(*
Nazwa:			FB_MoveRegister
Opis:			Blok przesuniecia rejestru formatek
Wersja:			v0.3 		
Data:			2018-11-16
Autor:			DP
Urzadzenia:		 
Konfiguracja:	
Info:
- Są dwa rejestry, wejściowy i wyjsciowy (struktury)
- Jezeli rejestr ma np. 6 elementów to za kazdym razem po wykryciu trigera program będzie
	1 wejściowy przesuwał na 1 wolny (nie ma formatki) wyjściowy
	kasował 1 rejestr wejściowy
	przesuwal rejetr wejsciowy 2 na 1(przeniesiony i skasowany), 3 na 2, 4 na 3, 5 na 4, 6 na 5 i kasowal 6wejsciowy
	tym sposobem po 6 trigerach caly rejestr wejsciowy powinien być na wyjsciowym
	np po 3 trigerach na wyjsciowym powinny byc zajete 1 do 3 i na wejsciowym 1 do 3
Błędy:
1 - nie wyszło z pętli for
2 - formatka już jest w rejestrze
Uwagi:
- 
Zmiany:
2018-09-18 Dodano sprawdzanie nasadek
2018-06-14 DP Pierwsza wersja
*)

FUNCTION_BLOCK FB_MoveRegister
VAR_INPUT
	bFirstCycle:BOOL;					//Pierwszy cykl, zeby na początku nie wykrywało zbocza opadającego
	bTrigger :BOOL;						// Przesuniecie tablicy o jeden
	tTriggerFilterTimeOn:TIME:=T#0MS;	// Czas filtrowania wejścia Trigger na załączenie
	tTriggerFilterTimeOff:TIME:=T#0MS;	// Czas filtrowania wejścia Trigger na wyłączenie
	bTriggerBottle :BOOL;				// Zapisywanie czy jest butelka czy nie (jezeli kontrola wlączona)
	bWithBottleControl: BOOL;			// Włączona opcja kontroli butelek
	bWithCapControl:BOOL;				// Wlaczona kontrola nasadek
	bWithFormControlTrigerCounter:BOOL;	// Jezeku na trigercontrol nie ma formatki do przesunięcia to stwórz nową
	bMoveOnlyToLastExitRegister:BOOL;	// Przepisuj rejestr wejściowy tylko na ostatni wyjściowy bez przesunięcia wyjściowego
	bMoveOnlyIfFormPresent:BOOL;		// Przepisuj tylko jak jest formatka
	bRotateEntranceRegisterBefore:BOOL;	// Najpierw przesuń rejestr wejściowy a następnie z niego zabierz
	bNoKeepTryingMove:BOOL;				// Dalej przepisuj jezeli nie ma miejsca
	bTriggerCap: BOOL;					// Truger wykrycia nasadki
	bReset :BOOL;						// Czyszczenie tablic
	iEntranceArrayElements :UINT; 		// Wartość koncowa tablicy
	iExitArrayElements :UINT; 			// Wartość koncowa tablicy
	bInvertWriting :BOOL;				// Wpisywanie odwrotne zamist z 1entrance na 1exit to 1entrance na 6exit	
	eClearPackageState :S_PackageState; // Czysty rejestr
END_VAR
VAR_IN_OUT
	bTriggerCounter :BOOL;		// Triger ktory jest kasowany
	eEntranceState :ARRAY [1..17] OF S_PackageState;	
	eExitState :ARRAY [1..17] OF S_PackageState;
	bKeepTryingMove :BOOL;		// Probuj dalej zapisać formatki aż się któraś zwolni
END_VAR

VAR_OUTPUT	
	bError :BOOL; 				// Błąd
	iError: UINT;				// Nr Błędu
	bTriggerDone :BOOL; 		// Wykonano przesunięcie
	bTriggerFilteredOUT:BOOL;	//Wyjscie przefiltrowanego sygnalu wejsciowego
END_VAR

VAR
	i:UINT;						// Zmienna w tablicy
	k:UINT;						// Pomocnicza zmienna do zapisywnia czy jest butelka
	rtbTrigger :R_TRIG;			// Reaguje na zbocze
	rtbTriggerBottle :R_TRIG;	// Reaguje na zbocze
	rtbReset :R_TRIG;			// Reaguje na zbocze
	TimerResetErrors :TON;		// Reset Błedu
	nFormCounter :UINT;					//Licznik formatek
	r1,r2:UINT;
	bBottlePresent: BOOL;				//Zmienna pomocnicza ze wykryto butelkę
	bCapPresent: BOOL;					//Zmienna pomocnicza ze wykryto butelkę
	j: UINT;
	tonTriggerFilterTimeOn: TON;
	bTriggerFiltered: BOOL;
	tofTriggerFilterTimeOff: TOF;
	tonTriggerFilterTimeBeforeTrigger: TON;
END_VAR

//Filtrowanie sygnału wejściowego
tofTriggerFilterTimeOff	(IN:=bTrigger, PT:=tTriggerFilterTimeOff);
tonTriggerFilterTimeOn	(IN:=tofTriggerFilterTimeOff.Q, PT:=tTriggerFilterTimeOn);
bTriggerFiltered 		:= tonTriggerFilterTimeOn.Q;
bTriggerFilteredOUT		:= bTriggerFiltered ;

//TRIGI I TIMERY
IF bWithBottleControl THEN
	rtbTrigger 	(CLK := NOT bTriggerFiltered, Q=>);
	rtbTriggerBottle 	(CLK := NOT bTriggerBottle, Q=>);
ELSIF bWithCapControl THEN
	rtbTrigger 	(CLK := NOT bTriggerFiltered, Q=>);
ELSE
	rtbTrigger 	(CLK := bTriggerFiltered, Q=>);
	rtbTriggerBottle 	(CLK := bTriggerBottle, Q=>);
END_IF

rtbReset 	(CLK := bReset, Q=>);
TimerResetErrors (IN:= bError, PT:=T#1000MS, Q=>);

//RESETOWANIE BLEDU
IF TimerResetErrors.Q THEN
	bError := FALSE;
END_IF

//KASOWANIE ZMIENNYCH
bTriggerDone := FALSE;

//JEZELI WLACZONO KONTROLE BUTELEK TO NADPISUJ REJESTR CZY JEST BUTELKA
IF bWithBottleControl AND bTrigger AND bTriggerBottle AND NOT bKeepTryingMove THEN //Jezeli od wykrycia formatki liczy TIMER i wykryło butelke to wpisz do rejestru że jest butelka
	eEntranceState[1].bBottlePresent := TRUE;
	eEntranceState[1].bFormPresent := TRUE;
	bBottlePresent := TRUE; // Wpisuje że jest butelka jezeli wystąpi sygnał podczas trwania czujnika formatki
ELSIF bWithBottleControl AND rtbTrigger.Q AND NOT bBottlePresent AND  NOT bKeepTryingMove AND bFirstCycle THEN
	eEntranceState[1].bBottlePresent := FALSE;
	eEntranceState[1].bFormPresent := TRUE; // jeżeli zanik czujnik formatki i nie było formatki to wpisz ze nie było butelki
END_IF
//JEZELI WLACZONO KONTROLE NASADEk TO NADPISUJ REJESTR CZY JEST BUTELKA 
(*IF bWithCapControl AND bTrigger AND bTriggerCap AND NOT bKeepTryingMove THEN //Jezeli od wykrycia formatki liczy TIMER i wykryło butelke to wpisz do rejestru że jest butelka
	eEntranceState[1].bCapPutted := TRUE;
	eEntranceState[1].bCapOK := TRUE; eEntranceState[1].bBottlePresent:= TRUE;//Zmiana nowa
	eEntranceState[1].bFormPresent := TRUE;
	bCapPresent := TRUE; // Wpisuje że jest butelka jezeli wystąpi sygnał podczas trwania czujnika formatki*)
	//ZMIANA LU 192
IF bWithCapControl AND bTriggerCap AND NOT bKeepTryingMove THEN //Jezeli od wykrycia formatki liczy TIMER i wykryło butelke to wpisz do rejestru że jest butelka
	eEntranceState[1].bCapPutted := TRUE;
	eEntranceState[1].bCapOK := TRUE; eEntranceState[1].bBottlePresent:= TRUE;//Zmiana nowa
	eEntranceState[1].bFormPresent := TRUE;
	bCapPresent := TRUE; // Wpisuje że jest butelka jezeli wystąpi sygnał podczas trwania czujnika formatki	
ELSIF bWithCapControl AND rtbTrigger.Q AND NOT bCapPresent AND  NOT bKeepTryingMove AND bFirstCycle THEN
	eEntranceState[1].bCapPutted := TRUE;
	eEntranceState[1].bCapOK:= FALSE;
	eEntranceState[1].bFormPresent := TRUE; // jeżeli zanik czujnik formatki i nie było formatki to wpisz ze nie było butelki
END_IF
//JEZELI WLACZONO SPRAWDZANIE FORMATEK Z TRIGERCOUNTER TO
IF bWithFormControlTrigerCounter  AND (bTriggerCounter OR rtbTrigger.Q) AND NOT bKeepTryingMove AND bFirstCycle THEN //Zmiena UBL50, tworz tez nowa jak Trigger
	eEntranceState[1].bFormPresent := TRUE;
END_IF



//PRZESUNIECIE
IF iEntranceArrayElements = iExitArrayElements AND bFirstCycle AND NOT bMoveOnlyToLastExitRegister THEN
	IF rtbTrigger.Q OR bKeepTryingMove OR bTriggerCounter THEN
		bTriggerCounter := FALSE; 
		bKeepTryingMove := FALSE;
		nFormCounter := 0;
		bBottlePresent:= bCapPresent  := FALSE; 
		IF NOT bInvertWriting THEN // Jezeli odwrotne wpisywanie
			FOR i := 1 TO iEntranceArrayElements DO
				IF  NOT eExitState[i].bFormPresent THEN  		// Jeżeli w rejestrze wyjściowym jest wolne miejsce to wpisz rejestr wejściowy
					eExitState[i] := eEntranceState[1];	// Wpisz do rejestru dane np z [1] Buffor do [1,2,3,4,5,6] Package
					eEntranceState[1]:=eClearPackageState;	// Czyszczenie pierwszego rejestru wejściowego
					k:=i;											// Przepisywanie zmiennej pomocniczej
					FOR i := 1 TO iEntranceArrayElements DO   				
						IF i = iEntranceArrayElements THEN
							eEntranceState[i]:=eClearPackageState;		  // Zerowanie ostatniego bo zostało przesuniete wszystko o 1
						ELSE													  // Przepisanie 2 do 1, 3 do 2, 4 do 3, 5 do 4, 6 do 5, zeruj 6
							eEntranceState[i] := eEntranceState[i+1]; // 2 do 1, 3 do 2,
							eEntranceState[i+1]:=eClearPackageState;		  // zeruj 2, 
						END_IF
					END_FOR
					bTriggerDone := TRUE;
					EXIT;
					bError := TRUE;
					iError := 1;
				ELSE
					nFormCounter := nFormCounter + 1;
					bError := TRUE;
					iError := 2;
				END_IF
			END_FOR
		ELSE
		
		//jezeli wybrano wpisywanie odwrotne
		
			FOR i := iEntranceArrayElements TO 1 BY -1 DO
				IF  NOT eExitState[i].bFormPresent THEN  		// Jeżeli w rejestrze wyjściowym jest wolne miejsce to wpisz rejestr wejściowy
					eExitState[i] := eEntranceState[1];	// Wpisz do rejestru dane np z [1] Buffor do [1,2,3,4,5,6] Package
					eEntranceState[1]:=eClearPackageState;	// Czyszczenie pierwszego rejestru wejściowego
					k:=i;											// Przepisywanie zmiennej pomocniczej
					FOR i := 1 TO iEntranceArrayElements DO   				
						IF i = iEntranceArrayElements THEN
							eEntranceState[i]:=eClearPackageState;		  // Zerowanie ostatniego bo zostało przesuniete wszystko o 1
						ELSE													  // Przepisanie 2 do 1, 3 do 2, 4 do 3, 5 do 4, 6 do 5, zeruj 6
							eEntranceState[i] := eEntranceState[i+1]; // 2 do 1, 3 do 2,
							eEntranceState[i+1]:=eClearPackageState;		  // zeruj 2, 
						END_IF
					END_FOR
					bTriggerDone := TRUE;
					EXIT;
					bError := TRUE;
					iError := 1;
				ELSE
					nFormCounter := nFormCounter + 1;
					bError := TRUE;
					iError := 2;
				END_IF
			END_FOR

		END_IF
		IF nFormCounter = iExitArrayElements THEN
		bKeepTryingMove:=NOT bNoKeepTryingMove;
		END_IF
	END_IF
ELSIF iEntranceArrayElements > iExitArrayElements AND bFirstCycle AND NOT bMoveOnlyToLastExitRegister THEN
	IF rtbTrigger.Q OR bKeepTryingMove OR bTriggerCounter THEN
		bTriggerCounter := FALSE; 
		bKeepTryingMove := FALSE;
		nFormCounter :=0;
		bBottlePresent := bCapPresent := FALSE; 
		IF NOT bInvertWriting THEN // Jezeli odwrotne wpisywanie
			FOR i := 1 TO iExitArrayElements DO
				IF  NOT eExitState[i].bFormPresent THEN  		// Jeżeli w rejestrze wyjściowym jest wolne miejsce to wpisz rejestr wejściowy
					eExitState[i] := eEntranceState[1];			// Wpisz do rejestru dane np z [1] Buffor do [1,2,3,4,5,6] Package
					eEntranceState[1]:=eClearPackageState;		// Czyszczenie pierwszego rejestru wejściowego
					k:=i;										// Przepisywanie zmiennej pomocniczej
					FOR i := 1 TO iEntranceArrayElements DO   				
						IF i = iEntranceArrayElements THEN
							eEntranceState[i]:=eClearPackageState;			// Zerowanie ostatniego bo zostało przesuniete wszystko o 1
						ELSE												// Przepisanie 2 do 1, 3 do 2, 4 do 3, 5 do 4, 6 do 5, zeruj 6
							IF NOT bMoveOnlyIfFormPresent THEN //ZMIANA LU192
								eEntranceState[i] := eEntranceState[i+1]; 		// 2 do 1, 3 do 2,
								eEntranceState[i+1]:=eClearPackageState;		// zeruj 2, 
							ELSE
								IF eEntranceState[i+1] .bFormPresent THEN
									eEntranceState[i] := eEntranceState[i+1]; 		// 2 do 1, 3 do 2,
									eEntranceState[i+1]:=eClearPackageState;		// zeruj 2, 	
								END_IF
							END_IF
						END_IF
					END_FOR
					bTriggerDone := TRUE;
					EXIT; 
					bError := TRUE;
					iError := 3;
				ELSE
					nFormCounter := nFormCounter + 1;
					bError := TRUE;
					iError := 4;
				END_IF
			END_FOR
		ELSE
			FOR i := iExitArrayElements TO 1 BY -1 DO
				IF  NOT eExitState[i].bFormPresent THEN  		// Jeżeli w rejestrze wyjściowym jest wolne miejsce to wpisz rejestr wejściowy
					eExitState[i] := eEntranceState[1];			// Wpisz do rejestru dane np z [1] Buffor do [1,2,3,4,5,6] Package
					eEntranceState[1]:=eClearPackageState;		// Czyszczenie pierwszego rejestru wejściowego
					k:=i;										// Przepisywanie zmiennej pomocniczej
					FOR i := 1 TO iEntranceArrayElements DO   				
						IF i = iEntranceArrayElements THEN
							eEntranceState[i]:=eClearPackageState;			// Zerowanie ostatniego bo zostało przesuniete wszystko o 1
						ELSE												// Przepisanie 2 do 1, 3 do 2, 4 do 3, 5 do 4, 6 do 5, zeruj 6
							eEntranceState[i] := eEntranceState[i+1]; 		// 2 do 1, 3 do 2,
							eEntranceState[i+1]:=eClearPackageState;		// zeruj 2, 
						END_IF
					END_FOR
					bTriggerDone := TRUE;
					EXIT;
					bError := TRUE;
					iError := 3;
				ELSE
					nFormCounter := nFormCounter + 1;
					bError := TRUE;
					iError := 4;
				END_IF
			END_FOR
		END_IF
	
		IF nFormCounter = iExitArrayElements THEN
			bKeepTryingMove:=NOT bNoKeepTryingMove;									
		END_IF																	
	END_IF
ELSIF iEntranceArrayElements < iExitArrayElements AND bFirstCycle AND NOT bMoveOnlyToLastExitRegister THEN
		IF rtbTrigger.Q OR bKeepTryingMove OR bTriggerCounter THEN
		bTriggerCounter := FALSE; 
		bKeepTryingMove := FALSE;
		nFormCounter := 0;
		(*Do testów - jeszcze raz nadpisz jakby czujniki były przestawione LU205*)	
		IF bCapPresent THEN		
			eEntranceState[1].bCapPutted := TRUE;
			eEntranceState[1].bCapOK := TRUE; eEntranceState[1].bBottlePresent:= TRUE;//Zmiana nowa
			eEntranceState[1].bFormPresent := TRUE;
		END_IF
		(*Koniec Do testów - jeszcze raz nadpisz jakby czujniki były przestawione*)

		bBottlePresent := bCapPresent  := FALSE; 
		IF NOT bInvertWriting AND NOT bRotateEntranceRegisterBefore THEN // Jezeli odwrotne wpisywanie
			FOR i := 1 TO iExitArrayElements DO
				IF  NOT eExitState[i].bFormPresent THEN  		// Jeżeli w rejestrze wyjściowym jest wolne miejsce to wpisz rejestr wejściowy
					eExitState[i] := eEntranceState[1];			// Wpisz do rejestru dane np z [1] Buffor do [1,2,3,4,5,6] Package
					eEntranceState[1]:=eClearPackageState;		// Czyszczenie pierwszego rejestru wejściowego
					k:=i;										// Przepisywanie zmiennej pomocniczej
					FOR i := 1 TO iEntranceArrayElements DO   				
						IF i = iEntranceArrayElements THEN
							eEntranceState[i]:=eClearPackageState;			// Zerowanie ostatniego bo zostało przesuniete wszystko o 1
						ELSE												// Przepisanie 2 do 1, 3 do 2, 4 do 3, 5 do 4, 6 do 5, zeruj 6
							eEntranceState[i] := eEntranceState[i+1]; 		// 2 do 1, 3 do 2,
							eEntranceState[i+1]:= eClearPackageState;		// zeruj 2, 
						END_IF
					END_FOR
					bTriggerDone := TRUE;
					EXIT;
					bError := TRUE;
					iError := 5;
				ELSE
					nFormCounter := nFormCounter + 1;
					bError := TRUE;
					iError := 6;
				END_IF
			END_FOR
		ELSIF bInvertWriting AND NOT bRotateEntranceRegisterBefore THEN
			FOR i := iExitArrayElements TO 1 BY -1 DO
				IF  NOT eExitState[i].bFormPresent THEN  		// Jeżeli w rejestrze wyjściowym jest wolne miejsce to wpisz rejestr wejściowy
					eExitState[i] := eEntranceState[1];			// Wpisz do rejestru dane np z [1] Buffor do [1,2,3,4,5,6] Package
					eEntranceState[1]:=eClearPackageState;		// Czyszczenie pierwszego rejestru wejściowego
					k:=i;										// Przepisywanie zmiennej pomocniczej
					FOR i := 1 TO iEntranceArrayElements DO   				
						IF i = iEntranceArrayElements THEN
							eEntranceState[i]:=eClearPackageState;			// Zerowanie ostatniego bo zostało przesuniete wszystko o 1
						ELSE												// Przepisanie 2 do 1, 3 do 2, 4 do 3, 5 do 4, 6 do 5, zeruj 6
							eEntranceState[i] := eEntranceState[i+1]; 		// 2 do 1, 3 do 2,
							eEntranceState[i+1]:= eClearPackageState;		// zeruj 2, 
						END_IF
					END_FOR
					bTriggerDone := TRUE;
					EXIT;
					bError := TRUE;
					iError := 5;
				ELSE
					nFormCounter := nFormCounter + 1;
					bError := TRUE;
					iError := 6;
				END_IF
			END_FOR
		ELSIF NOT bInvertWriting AND bRotateEntranceRegisterBefore THEN //Opcja najpierw przepisz a potem zabierz 
			FOR i := 1 TO iExitArrayElements DO
				IF  NOT eExitState[i].bFormPresent THEN  		// Jeżeli w rejestrze wyjściowym jest wolne miejsce to wpisz rejestr wejściowy
																// Przepisywanie zmiennej pomocniczej
					FOR j := 1 TO iEntranceArrayElements DO   				
						IF j = iEntranceArrayElements THEN
							eEntranceState[j]:=eClearPackageState;			// Zerowanie ostatniego bo zostało przesuniete wszystko o 1
						ELSE												// Przepisanie 2 do 1, 3 do 2, 4 do 3, 5 do 4, 6 do 5, zeruj 6
							eEntranceState[j] := eEntranceState[j+1]; 		// 2 do 1, 3 do 2,
							eEntranceState[j+1]:= eClearPackageState;		// zeruj 2, 
						END_IF
					END_FOR
					
					eExitState[i] := eEntranceState[1];			// Wpisz do rejestru dane np z [1] Buffor do [1,2,3,4,5,6] Package
					eEntranceState[1]:=eClearPackageState;		// Czyszczenie pierwszego rejestru wejściowego
					k:=i;
					
					bTriggerDone := TRUE;
					EXIT;
					bError := TRUE;
					iError := 5;
				ELSE
					nFormCounter := nFormCounter + 1;
					bError := TRUE;
					iError := 6;
				END_IF
			END_FOR
		END_IF
		IF nFormCounter = iExitArrayElements THEN
			bKeepTryingMove:=NOT bNoKeepTryingMove;
		END_IF
	END_IF
ELSIF bMoveOnlyToLastExitRegister THEN //Opcja wpisywania z rejestru wejsciowego na ostatni wyjsciowy bez przesuwania wyjsciowego 
		IF rtbTrigger.Q OR bKeepTryingMove OR bTriggerCounter THEN
		bTriggerCounter := FALSE; 
		bKeepTryingMove := FALSE;
		nFormCounter := 0;
		
		(*Do testów - jeszcze raz nadpisz jakby czujniki były przestawione LU205*)	
		IF bCapPresent THEN		
			eEntranceState[1].bCapPutted := TRUE;
			eEntranceState[1].bCapOK := TRUE; eEntranceState[1].bBottlePresent:= TRUE;//Zmiana nowa
			eEntranceState[1].bFormPresent := TRUE;
		END_IF
		(*Koniec Do testów - jeszcze raz nadpisz jakby czujniki były przestawione*)					
		bBottlePresent := bCapPresent := FALSE; 
		
				IF  NOT bWithCapControl AND NOT eExitState[iExitArrayElements].bFormPresent AND NOT bRotateEntranceRegisterBefore THEN  	// Jeżeli w rejestrze wyjściowym jest wolne miejsce to wpisz rejestr wejściowy
					eExitState[iExitArrayElements] := eEntranceState[1];	// Wpisz do rejestru dane np z [1] Buffor do [1,2,3,4,5,6] Package
					eEntranceState[1]:=eClearPackageState;		// Czyszczenie pierwszego rejestru wejściowego
					k:=i;										// Przepisywanie zmiennej pomocniczej
					FOR i := 1 TO iEntranceArrayElements DO   				
						IF i = iEntranceArrayElements THEN
							eEntranceState[i]:=eClearPackageState;			// Zerowanie ostatniego bo zostało przesuniete wszystko o 1
						ELSE												// Przepisanie 2 do 1, 3 do 2, 4 do 3, 5 do 4, 6 do 5, zeruj 6
							eEntranceState[i] := eEntranceState[i+1]; 		// 2 do 1, 3 do 2,
							eEntranceState[i+1]:= eClearPackageState;		// zeruj 2, 
						END_IF
					END_FOR
					bTriggerDone := TRUE;
					
					bError := TRUE;
					iError := 5;
				ELSIF bWithCapControl AND NOT bRotateEntranceRegisterBefore THEN //TUTAJ DODAŁEM
					eExitState[iExitArrayElements] := eEntranceState[1];	// Wpisz do rejestru dane np z [1] Buffor do [1,2,3,4,5,6] Package
					eEntranceState[1]:=eClearPackageState;		// Czyszczenie pierwszego rejestru wejściowego
					k:=i;										// Przepisywanie zmiennej pomocniczej
(*zmiana dp-1*)		FOR i := 1 TO iEntranceArrayElements DO   			
						IF i = iEntranceArrayElements THEN
							eEntranceState[i]:=eClearPackageState;			// Zerowanie ostatniego bo zostało przesuniete wszystko o 1
						ELSE												// Przepisanie 2 do 1, 3 do 2, 4 do 3, 5 do 4, 6 do 5, zeruj 6
							eEntranceState[i] := eEntranceState[i+1]; 		// 2 do 1, 3 do 2,
							eEntranceState[i+1]:= eClearPackageState;		// zeruj 2, 
						END_IF
					END_FOR
					bTriggerDone := TRUE;
					
				(*NEW*)	
				ELSIF NOT bInvertWriting AND bRotateEntranceRegisterBefore THEN //Opcja najpierw przepisz a potem zabierz 

							FOR j := 1 TO iEntranceArrayElements DO   				
								IF j = iEntranceArrayElements THEN
									eEntranceState[j]:=eClearPackageState;			// Zerowanie ostatniego bo zostało przesuniete wszystko o 1
								ELSE												// Przepisanie 2 do 1, 3 do 2, 4 do 3, 5 do 4, 6 do 5, zeruj 6
									eEntranceState[j] := eEntranceState[j+1]; 		// 2 do 1, 3 do 2,
									eEntranceState[j+1]:= eClearPackageState;		// zeruj 2, 
								END_IF
							END_FOR
							eExitState[iExitArrayElements] := eEntranceState[1];	// Wpisz do rejestru dane np z [1] Buffor do [1,2,3,4,5,6] Package
							eEntranceState[1]:=eClearPackageState;					// Czyszczenie pierwszego rejestru wejściowego
							bTriggerDone := TRUE;
							bError := TRUE;
							iError := 5;
		
				ELSE
					nFormCounter := nFormCounter + 1;
					bError := TRUE;
					iError := 6;
				END_IF				
				
			IF nFormCounter = 1 THEN
				bKeepTryingMove:=NOT bNoKeepTryingMove;
			END_IF
		END_IF
END_IF	


//CZYSZCZENIE REJESTRU WEJSCIOWEGO
IF rtbReset.Q THEN
	FOR r1 := 1 TO iEntranceArrayElements DO
		eEntranceState[r1] := eClearPackageState;
	END_FOR
	FOR r2 := 1 TO iExitArrayElements DO
		eExitState[r2] := eClearPackageState;
	END_FOR
	bKeepTryingMove :=FALSE;
	bTriggerDone := FALSE;
	bTriggerCounter := FALSE; 
	nFormCounter := 0;
	bBottlePresent := bCapPresent := FALSE; 
	bError := FALSE;
	iError := 0;
END_IF

END_FUNCTION_BLOCK

(* stored: Version 1.1.0.1, ProductVersion 3.1.4026.13, FileIdentifier f984fe407f20204899cafed5b34901bfef2a62a0, FileSignature 941aed538e385ad0ebbdf01b80e0cc81b07a8a4f44069327e620a31a6baabe852f7843a74683a1442745ba0e2d63d8797d30573f080eea1685ba2c00d14043fb605733171bb772aae057e9b192529598264d349705d3dd1818427cd255e0abf25bb56e1a4e68af4896bb7f30096b637f882072d61c3629694593e80f58b6d38a56dd1a365b0f6e9d31f3a019bad90123d8b49578248053ef58ae90cf654efe8db825a72e04d1b70b1832554775ec5bb7ad882ff532e7a32f31051418bdf521a820e458e2e17e7c6e2f84ba1be691e1ca1d465a4229b4125965c0ebd087efb9f12919a22f9668ad27b871aa640ea205c8f04cc33473e311165095ece2adeca152
   POU FB_MoveRegister: Id {1909d49d-a9cc-438b-ba4f-b1649b3b9513}, SpecialFunc None *)
